Fanuc KAREL source: kb00090.KL

-- PROVISIONAL review KL for V940-1; original PC SHA256 82c6d7dc124dd59e1cd681f6cc9fcd0dd06a15ce45ab48f8180901a5b2894a98
-- Incomplete behavior may be omitted. Consult companion uncertainty JSON. Do not deploy.
PROGRAM KB00090
%NOLOCKGROUP
BEGIN
  -- V9_ZERO_TABLE_METADATA_HINT layout=0002_ascii; no indexed target words; source/name/runtime held
  -- UNRESOLVED_PC offsets 5-12; opcodes 9D,23
  -- UNRESOLVED_PC offsets 17-24; opcodes 9D,23
  -- UNRESOLVED_PC offsets 29-36; opcodes 9D,23
  -- UNRESOLVED_PC offsets 41-52; opcodes 2E,23
  -- UNRESOLVED_PC offsets 57-64; opcodes 9D,23
  -- UNRESOLVED_PC offsets 69-103; opcodes 27,22,22,22,22,22,31
  -- UNRESOLVED_PC offsets 108-112; opcodes 7F
END KB00090
